FUNCTION_BLOCK DriveSim EXTENDS TcoCore.TcoComponent IMPLEMENTS IDrive
VAR
    {attribute addProperty Name "<#Current position#>"}
    _position : LREAL;
END_VAR
VAR
    {attribute addProperty Name "<#Move absolute#>"}
    {attribute addProperty ToolTip "<#Moves the drive to absolute position given by parameter 'Target Position'#>"}
    _moveAbsoluteTask : DriveSimMoveAbsoluteTask(THIS^);
END_VAR

_moveAbsoluteTask(_drive := THIS^);

METHOD MoveAbsolute : TcoCore.ITcoTaskStatus
VAR_INPUT
    TargetPosition : LREAL;
END_VAR
_moveAbsoluteTask.TargetPosition := TargetPosition;
MoveAbsolute := _moveAbsoluteTask.Invoke();
END_METHOD

PROPERTY MoveAbsoluteTask : REFERENCE TO DriveSimMoveAbsoluteTask
GET
MoveAbsoluteTask REF= _moveAbsoluteTask;
END_GET
END_PROPERTY

PROPERTY Position : LREAL
GET
Position := _position;
END_GET
SET
_position := Position;
END_SET
END_PROPERTY

(*~
    <docu>
        <summary>
            Restores this instance to the Ready state. Can be called explicitly or from within one of the restore mechanisms.
        </summary>
    </docu>
~*)
METHOD Restore : ITcoRestorable
END_METHOD

(*~
    <docu>
        <summary>
            Custom service (manual, maintenance) logic.
            This method must be implemented in derived class.
        </summary>
    </docu>
~*)
METHOD PROTECTED ServiceMode
END_METHOD

END_FUNCTION_BLOCK

(* stored: Version 1.1.0.1, ProductVersion 3.1.4024.9
   POU DriveSim: Id {268333eb-fb89-4342-a1df-991907c3378e}, SpecialFunc None
   Method MoveAbsolute: Id {f73759c6-de9b-49ed-83e9-08090b234b0f}
   Property MoveAbsoluteTask: Id {523daa0d-a2eb-4f3e-95b5-945fa86dbbad}
   Get Get: Id {4ae57316-fc76-4112-ad1f-822c3c895b6c}
   Property Position: Id {21e50bee-72b1-4176-b263-6166c4cf89fd}
   Get Get: Id {6fe391a0-8205-4811-9253-7d81a1d28378}
   Set Set: Id {abd4498c-ca56-498d-a5a7-89b2b0c47016}
   Method Restore: Id {8996e689-e19d-4f58-87af-5ad072d65536}
   Method ServiceMode: Id {2b5a6043-3c89-4c07-925b-b7c03231b81f} *)
